Xinje XDPPro project, PLC1: XDH-60T4 (software 3.7.4b 2021-06-17)

PROGRAM Ladder

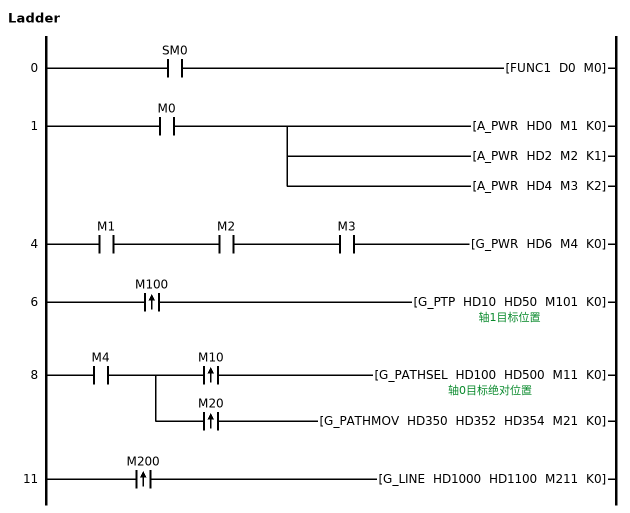
LD     SM0
FUNC1  D0 M0
LD     M0
A_PWR  HD0 M1 K0
A_PWR  HD2 M2 K1
A_PWR  HD4 M3 K2
LD     M1
AND    M2
AND    M3
G_PWR  HD6 M4 K0
LDP    M100
G_PTP  HD10 HD50 M101 K0	; 轴1目标位置
LD     M4
MPS
ANDP   M10
G_PATHSEL HD100 HD500 M11 K0	; 轴0目标绝对位置
MPP
ANDP   M20
G_PATHMOV HD350 HD352 HD354 M21 K0
LDP    M200
G_LINE HD1000 HD1100 M211 K0

COMMENTS (devices not used above)
D20444	轴3当前位置
D20244	轴2当前位置
HD200	轴1目标绝对位置
D20044	轴1当前位置
HD14	轴2目标位置
HD18	轴3目标位置

C FUNCTION BLOCK func1.fcb
/*************************************************************************
   FunctionBlockName:  FUNC1
   Version:            1.0.0
   Author:             
   UpdateTime:         2021-08-21 17:10:53
   Comment:            
			
**************************************************************************/
void FUNC1( WORD W , BIT B )
{
#define SysRegAddr_HD_D_HM_M
#define DFHD *(FP64*)&HD

HD[100] = 3;
HD[101] = 0;

HD[110] = 1;
HD[112] = 1;
HD[113] = 0;
DFHD[116] = 100000;
DFHD[120] = 100000;
DFHD[124] = 0;
DFHD[164] = 20000;

HD[170] = 2;
HD[172] = 0;
HD[173] = 0;
DFHD[176] = 200000;
DFHD[180] = 150000;
DFHD[184] = 0;
DFHD[224] = 20000;

HD[230] = 3;
HD[232] = 200;
HD[233] = 0;


}